function_block FB_Syntax_StweepDisable  
var
    nA : INT;  
    nB      : int;
end_var

nA := 1;


{stweep.disable}
nA := 99;
nB := 88;
{stweep.enable}
(* @stweep.disable *)
nA := 77;
(* @stweep.enable *)  


nB := 2;

END_FUNCTION_BLOCK

(* stored: Version 1.1.0.1, ProductVersion 3.1.4024.16
   POU FB_Syntax_StweepDisable: Id {c4547a05-dd71-43d1-afc7-284783fab01a}, SpecialFunc None *)
